% RSLogix 500 project lab 10 prelab.RSS, saved by version 8.30.00.16 %
PROJECT "UNTITLED"    % processor: MicroLogix 1000 %

PROGRAM FILES
  LAD 2 "MAIN_PROG"  10 rungs
  LAD 3 "USER_FAULT"  1 rungs
  LAD 4 "HSC_INT"  1 rungs
  LAD 5 "STI_INT"  1 rungs
  LAD 6, 7, 8, 9, 10, 11, 12, 13, 14, 15, 16: only END

DATA FILES
  O0 OUTPUT  1 elements
  I1 INPUT  2 elements
  S2 STATUS  33 elements
  B3 BINARY  32 elements
  T4 TIMER  40 elements
  C5 COUNTER  32 elements
  R6 CONTROL  16 elements
  N7 INTEGER  105 elements

LADDER 2 "MAIN_PROG"
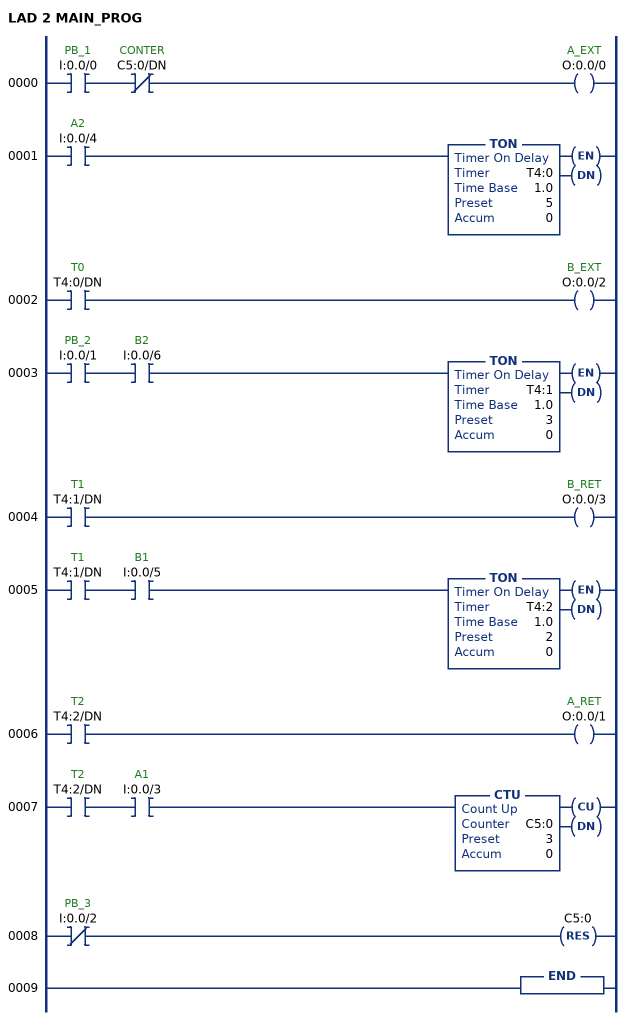
% Rung: 0 %  % edit flag set %
SOR XIC I:0.0/0 XIO C5:0/DN OTE O:0.0/0 EOR
%   I:0.0/0  PB_1 %
%   C5:0/DN  CONTER %
%   O:0.0/0  A_EXT %
% Rung: 1 %  % edit flag set %
SOR XIC I:0.0/4 TON T4:0 1.0 5 0 EOR
%   I:0.0/4  A2 %
% Rung: 2 %  % edit flag set %
SOR XIC T4:0/DN OTE O:0.0/2 EOR
%   T4:0/DN  T0 %
%   O:0.0/2  B_EXT %
% Rung: 3 %  % edit flag set %
SOR XIC I:0.0/1 XIC I:0.0/6 TON T4:1 1.0 3 0 EOR
%   I:0.0/1  PB_2 %
%   I:0.0/6  B2 %
% Rung: 4 %  % edit flag set %
SOR XIC T4:1/DN OTE O:0.0/3 EOR
%   T4:1/DN  T1 %
%   O:0.0/3  B_RET %
% Rung: 5 %  % edit flag set %
SOR XIC T4:1/DN XIC I:0.0/5 TON T4:2 1.0 2 0 EOR
%   T4:1/DN  T1 %
%   I:0.0/5  B1 %
% Rung: 6 %  % edit flag set %
SOR XIC T4:2/DN OTE O:0.0/1 EOR
%   T4:2/DN  T2 %
%   O:0.0/1  A_RET %
% Rung: 7 %  % edit flag set %
SOR XIC T4:2/DN XIC I:0.0/3 CTU C5:0 3 0 EOR
%   T4:2/DN  T2 %
%   I:0.0/3  A1 %
% Rung: 8 %  % edit flag set %
SOR XIO I:0.0/2 RES C5:0 EOR
%   I:0.0/2  PB_3 %
% Rung: 9 %
SOR END EOR
